// TwinCAT 3 PLC project HomeControl
// ProgramVersion: 3.1.4023.0
// libraries:
//   Tc2_Standard, * (Beckhoff Automation GmbH)
//   Tc2_System, * (Beckhoff Automation GmbH)
//   Tc3_Module, * (Beckhoff Automation GmbH)
// project tree:
//   / PlcTask.TcTTO
//   POUs/Communication/ESPNow/ FB_ESPNow.TcPOU
//   POUs/Communication/MQTT/ FB_MQTT.TcPOU
//   POUs/Communication/SerialCom/ FB_SerialCom.TcPOU
//   POUs/Device/AirConditioner/ FB_AirConditionerBase.TcPOU
//   POUs/Device/AirConditioner/Mitsubishi/ FB_AC_Mitsubishi.TcPOU
//   POUs/Device/AirConditioner/Siemens/ FB_AC_Siemens.TcPOU, ST_AC_Siemens.TcDUT
//   POUs/Device/ FB_Device.TcPOU
//   POUs/Device/Sensors/BinarySensor/ FB_BinarySensor.TcPOU
//   POUs/Device/Sensors/ FB_SensorBase.TcPOU
//   POUs/Device/Sensors/TemparatureSensor/ FB_TemperatureSensor.TcPOU
//   POUs/ESP01/ FB_ESP01.TcPOU
//   POUs/ESP8266/ FB_ESP8266.TcPOU, FB_SystemManager.TcPOU
//   POUs/ MAIN.TcPOU
// real-time tasks:
//   TASK PlcTask: cycle T#10ms, priority 20, ADS port 350

CONFIGURATION HomeControl
    RESOURCE PLC ON TwinCAT3
        TASK PlcTask(INTERVAL := T#10ms, PRIORITY := 20);
        PROGRAM MAIN WITH PlcTask : MAIN;
    END_RESOURCE
END_CONFIGURATION

// ---- POUs/Device/AirConditioner/Siemens/ST_AC_Siemens.TcDUT
TYPE ST_AC_Siemens :
STRUCT
	Protocol: STRING;
	Model : STRING;
END_STRUCT
END_TYPE

// ---- POUs/MAIN.TcPOU
PROGRAM MAIN
VAR
	fbESP01 : FB_ESP01;
	fbESP8266 : FB_ESP8266;
END_VAR

//Test
(*
1- fbESP8266 içindeki fbSerialCom.readTest değişkenini trueya çekerse register olurlar.

*)
fbESP8266();

END_PROGRAM

// ---- POUs/ESP01/FB_ESP01.TcPOU
FUNCTION_BLOCK FB_ESP01
VAR_INPUT
END_VAR
VAR_OUTPUT
END_VAR
VAR
	fbESPNow : FB_ESPNow;
	fbSerialCom : FB_SerialCom; 
END_VAR

END_FUNCTION_BLOCK

// ---- POUs/Communication/ESPNow/FB_ESPNow.TcPOU
FUNCTION_BLOCK FB_ESPNow
VAR_INPUT
END_VAR
VAR_OUTPUT
END_VAR
VAR
END_VAR

END_FUNCTION_BLOCK

// ---- POUs/Communication/SerialCom/FB_SerialCom.TcPOU
FUNCTION_BLOCK FB_SerialCom
VAR_INPUT
END_VAR
VAR_OUTPUT
END_VAR
VAR
	macAddrTest: STRING := '16';
	messageTest: STRING:= 'hasan';
	lenTest: INT:=5;
	readTest: BOOL;
END_VAR

PROPERTY length : int
GET
length := lenTest;
END_GET
SET
END_SET
END_PROPERTY

PROPERTY macAddr : string
GET
macAddr := macAddrTest;
END_GET
SET
END_SET
END_PROPERTY

PROPERTY message : string
GET
message := messageTest;
END_GET
SET
END_SET
END_PROPERTY

METHOD read : BOOL
VAR_INPUT
END_VAR
IF readTest THEN
	read := TRUE;
	readTest := FALSE;
END_IF
END_METHOD

METHOD write : BOOL
VAR_INPUT
	message: STRING;
END_VAR
END_METHOD

END_FUNCTION_BLOCK

// ---- POUs/ESP8266/FB_ESP8266.TcPOU
FUNCTION_BLOCK FB_ESP8266
VAR_INPUT
END_VAR
VAR_OUTPUT
END_VAR
VAR
	fbSystemManager : FB_SystemManager;
	fbMQTT :FB_MQTT;
	fbSerialCom : FB_SerialCom; 
	MqttMessageAvailable: BOOL;
	
	//testDevices
	fbAcMitsubishi: FB_AC_Mitsubishi;
	fbDoorSensor: FB_BinarySensor;
END_VAR

IF InitModule() THEN
	fbSystemManager.ExecuteDevices();
	IF fbSerialCom.read() THEN
		DeserializeMessage(fbSerialCom.macAddr,fbSerialCom.message,fbSerialCom.length);
	END_IF	
END_IF

METHOD DeserializeMessage : BOOL
VAR_INPUT
	MacAddr: STRING;
	message : STRING;
	length: INT;
END_VAR
VAR
	device : POINTER TO FB_Device;
END_VAR
// Deserialize Message
device := fbSystemManager.FilterDeviceMacAddr(MacAddr);
IF device<> 0 THEN
	device^.HandleMessage(message);
END_IF
END_METHOD

METHOD InitModule : BOOL
VAR_INPUT
END_VAR
VAR_INST
	idx: INT;
END_VAR
case idx of
	0:
		fbSerialCom.write('InitBroadcast');
		idx := 1;
	1:
		IF fbSerialCom.read()THEN
			fbAcMitsubishi.Id := 1;
			fbAcMitsubishi.MacAddr:='16';
			fbAcMitsubishi.Name:= 'Klima';
			fbSystemManager.registerDevice(fbAcMitsubishi);
			
			fbDoorSensor.Id := 2;
			fbDoorSensor.MacAddr:='26';
			fbDoorSensor.Name:= 'Kapi Sensor';
			fbSystemManager.registerDevice(fbDoorSensor);
			idx := 2;
		END_IF
	2:
		InitModule := TRUE;
END_CASE
END_METHOD

METHOD SerializeMessage : BOOL
VAR_INPUT
	topic: STRING;
	payload: STRING;
	length: INT;
END_VAR
//convert json and send
fbSerialCom.write('test');
END_METHOD

END_FUNCTION_BLOCK

// ---- POUs/ESP8266/FB_SystemManager.TcPOU
FUNCTION_BLOCK FB_SystemManager
VAR_INPUT
END_VAR
VAR_OUTPUT
END_VAR
VAR
	Devices : ARRAY [1..100] OF POINTER TO FB_Device;
	nRegisteredDevice :INT;
END_VAR

METHOD ExecuteDevices : BOOL
VAR
	idx: INT;
END_VAR
FOR idx :=1 TO nRegisteredDevice DO
	Devices[idx]^.Execute();
END_FOR
END_METHOD

METHOD FilterDeviceMacAddr : POINTER TO FB_Device;
VAR_INPUT
	macAdr: STRING;
END_VAR

VAR
	idx: INT;
END_VAR
FOR idx := 1 TO nRegisteredDevice DO
	IF Devices[idx]^.MacAddr = macAdr THEN
		FilterDeviceMacAddr := Devices[idx];
		RETURN;
	END_IF
END_FOR
END_METHOD

PROPERTY NumberOfRegisteredDevice : int
GET
END_GET
END_PROPERTY

METHOD registerDevice : BOOL
VAR_INPUT
	pDevice : REFERENCE TO FB_Device;
END_VAR
nRegisteredDevice := nRegisteredDevice + 1;
Devices[nRegisteredDevice] := ADR(pDevice);

ADSLOGSTR(msgCtrlMask := ADSLOG_MSGTYPE_ERROR, msgFmtStr := 'Registered Instance: %s', strArg := pDevice.Name);
END_METHOD

METHOD UnregisterDevice : BOOL
VAR_INPUT
END_VAR
END_METHOD

END_FUNCTION_BLOCK

// ---- POUs/Device/FB_Device.TcPOU
FUNCTION_BLOCK ABSTRACT FB_Device
VAR_INPUT
END_VAR
VAR_OUTPUT
END_VAR
VAR
	_id: INT;
	_macAddr: STRING;
	_name: STRING;
END_VAR

METHOD Execute : BOOL
VAR_INPUT
END_VAR
END_METHOD

METHOD ABSTRACT HandleMessage : BOOL
VAR_INPUT
	message :STRING;
END_VAR
END_METHOD

PROPERTY Id : int
GET
Id := _id;
END_GET
SET
_id := Id;
END_SET
END_PROPERTY

PROPERTY MacAddr : String
GET
MacAddr := _macAddr;
END_GET
SET
_macAddr := MacAddr;
END_SET
END_PROPERTY

PROPERTY Name : String
GET
Name := _name;
END_GET
SET
_name := Name;
END_SET
END_PROPERTY

METHOD SendMessage : BOOL
VAR_INPUT
END_VAR
END_METHOD

END_FUNCTION_BLOCK

// ---- POUs/Communication/MQTT/FB_MQTT.TcPOU
FUNCTION_BLOCK FB_MQTT
VAR_INPUT
END_VAR
VAR_OUTPUT
END_VAR
VAR
END_VAR

END_FUNCTION_BLOCK

// ---- POUs/Device/AirConditioner/Mitsubishi/FB_AC_Mitsubishi.TcPOU
FUNCTION_BLOCK FB_AC_Mitsubishi EXTENDS FB_AirConditionerBase
VAR_INPUT
END_VAR
VAR_OUTPUT
END_VAR
VAR
END_VAR

METHOD HandleMessage : BOOL
VAR_INPUT
	message :STRING;
END_VAR
IF message='turnedOff' THEN
	ADSLOGSTR(msgCtrlMask := ADSLOG_MSGTYPE_ERROR, msgFmtStr := 'Mitsubishi Air Conditioner Turned Off', strArg := '');
END_IF
END_METHOD

END_FUNCTION_BLOCK

// ---- POUs/Device/AirConditioner/FB_AirConditionerBase.TcPOU
FUNCTION_BLOCK ABSTRACT FB_AirConditionerBase EXTENDS FB_Device
VAR_INPUT
END_VAR
VAR_OUTPUT
END_VAR
VAR
END_VAR

METHOD TurnOff : BOOL
VAR_INPUT
END_VAR
END_METHOD

METHOD TurnOn : BOOL
VAR_INPUT
END_VAR
END_METHOD

END_FUNCTION_BLOCK

// ---- POUs/Device/Sensors/BinarySensor/FB_BinarySensor.TcPOU
FUNCTION_BLOCK FB_BinarySensor EXTENDS FB_SensorBase
VAR_INPUT
END_VAR
VAR_OUTPUT
END_VAR
VAR
END_VAR

METHOD HandleMessage : BOOL
VAR_INPUT
	message :STRING;
END_VAR
IF message='1' THEN
	ADSLOGSTR(msgCtrlMask := ADSLOG_MSGTYPE_ERROR, msgFmtStr := 'Door Opened', strArg := '');
END_IF
END_METHOD

END_FUNCTION_BLOCK

// ---- POUs/Device/Sensors/FB_SensorBase.TcPOU
FUNCTION_BLOCK FB_SensorBase EXTENDS FB_Device
VAR_INPUT
END_VAR
VAR_OUTPUT
END_VAR
VAR
END_VAR

METHOD  HandleMessage : BOOL
VAR_INPUT
	message :STRING;
END_VAR
END_METHOD

END_FUNCTION_BLOCK

// ---- POUs/Device/AirConditioner/Siemens/FB_AC_Siemens.TcPOU
FUNCTION_BLOCK FB_AC_Siemens EXTENDS FB_AirConditionerBase
VAR_INPUT
END_VAR
VAR_OUTPUT
END_VAR
VAR
END_VAR

METHOD Execute : BOOL
VAR_INPUT
END_VAR
VAR
	TurnOnCommand: BOOL;
	TurnOffCommand: BOOL;
END_VAR
PublishDeviceData();
END_METHOD

METHOD HandleMessage : BOOL
VAR_INPUT
	message: STRING;
END_VAR
VAR
	TurnOnCommand: BOOL;
	TurnOffCommand: BOOL;
END_VAR
IF TurnOffCommand THEN
	TurnOff();
ELSIF TurnOnCommand THEN
	TurnOn();
END_IF
END_METHOD

METHOD PublishDeviceData : BOOL
VAR_INPUT
END_VAR
END_METHOD

METHOD TurnOff : BOOL
VAR_INPUT
END_VAR
END_METHOD

METHOD TurnOn : BOOL
VAR_INPUT
END_VAR
//turn on Struct created
END_METHOD

END_FUNCTION_BLOCK

// ---- POUs/Device/Sensors/TemparatureSensor/FB_TemperatureSensor.TcPOU
FUNCTION_BLOCK FB_TemperatureSensor
VAR_INPUT
END_VAR
VAR_OUTPUT
END_VAR
VAR
END_VAR

END_FUNCTION_BLOCK
